// TwinCAT 3 PLC project PLCSim
// ProgramVersion: 3.1.4026.21
// libraries:
//   Tc2_Standard, * (Beckhoff Automation GmbH)
//   Tc2_System, * (Beckhoff Automation GmbH)
//   Tc3_Module, * (Beckhoff Automation GmbH)
//   VisuSymbols,newest,System
// project tree:
//   / GlobalTextList.TcGTLO, PlcTask.TcTTO (not stored), Visualization Manager.TcVMO (not stored)
//   POUs/ MAIN.TcPOU
//   VISUs/ Visualization.TcVIS
// real-time tasks:
//   TASK PlcTask: cycle T#30ms, priority 20, ADS port 350
// variable links:
//   PLCSim/PLCSim Instance <-> PLCStudent/PLCStudent Instance
//     PlcTask Inputs/MAIN.ixDrillDown <-> PlcTask Outputs/ControlFBD.qxDrillDown
//     PlcTask Inputs/MAIN.ixDrillUp <-> PlcTask Outputs/ControlFBD.qxDrillUp
//     PlcTask Inputs/MAIN.ixLampEmStopOk <-> PlcTask Outputs/ControlFBD.qxLampEmStopOk
//     PlcTask Inputs/MAIN.ixLampHomePos <-> PlcTask Outputs/ControlFBD.qxLampHomePos
//     PlcTask Inputs/MAIN.ixLampSafetyOk <-> PlcTask Outputs/ControlFBD.qxLampSafetyOk
//     PlcTask Inputs/MAIN.ixLampStarted <-> PlcTask Outputs/ControlFBD.qxLampStarted
//     PlcTask Inputs/MAIN.ixSliderAin <-> PlcTask Outputs/ControlFBD.qxSliderAin
//     PlcTask Inputs/MAIN.ixSliderAout <-> PlcTask Outputs/ControlFBD.qxSliderAout
//     PlcTask Inputs/MAIN.ixSliderBin <-> PlcTask Outputs/ControlFBD.qxSliderBin
//     PlcTask Inputs/MAIN.ixSliderBout <-> PlcTask Outputs/ControlFBD.qxSliderBout
//     PlcTask Outputs/MAIN.qxAuto <-> PlcTask Inputs/ControlFBD.ixAuto
//     PlcTask Outputs/MAIN.qxBtn1EmStopOk <-> PlcTask Inputs/ControlFBD.ixBtn1EmStopOk
//     PlcTask Outputs/MAIN.qxBtn2EmStopOk <-> PlcTask Inputs/ControlFBD.ixBtn2EmStopOk
//     PlcTask Outputs/MAIN.qxBtnAin <-> PlcTask Inputs/ControlFBD.ixBtnAin
//     PlcTask Outputs/MAIN.qxBtnAout <-> PlcTask Inputs/ControlFBD.ixBtnAout
//     PlcTask Outputs/MAIN.qxBtnBin <-> PlcTask Inputs/ControlFBD.ixBtnBin
//     PlcTask Outputs/MAIN.qxBtnBout <-> PlcTask Inputs/ControlFBD.ixBtnBout
//     PlcTask Outputs/MAIN.qxBtnDrillIn <-> PlcTask Inputs/ControlFBD.ixBtnDrillIn
//     PlcTask Outputs/MAIN.qxBtnDrillOut <-> PlcTask Inputs/ControlFBD.ixBtnDrillOut
//     PlcTask Outputs/MAIN.qxBtnReset <-> PlcTask Inputs/ControlFBD.ixBtnReset
//     PlcTask Outputs/MAIN.qxButtonStart <-> PlcTask Inputs/ControlFBD.ixButtonStart
//     PlcTask Outputs/MAIN.qxButtonStop <-> PlcTask Inputs/ControlFBD.ixButtonStop
//     PlcTask Outputs/MAIN.qxDrillDown <-> PlcTask Inputs/ControlFBD.ixDrillDown
//     PlcTask Outputs/MAIN.qxDrillUp <-> PlcTask Inputs/ControlFBD.ixDrillUp
//     PlcTask Outputs/MAIN.qxSafety1StopOk <-> PlcTask Inputs/ControlFBD.ixSafety1StopOk
//     PlcTask Outputs/MAIN.qxSafety2StopOk <-> PlcTask Inputs/ControlFBD.ixSafety2StopOk
//     PlcTask Outputs/MAIN.qxSliderAin <-> PlcTask Inputs/ControlFBD.ixSliderAin
//     PlcTask Outputs/MAIN.qxSliderAout <-> PlcTask Inputs/ControlFBD.ixSliderAout
//     PlcTask Outputs/MAIN.qxSliderBin <-> PlcTask Inputs/ControlFBD.ixSliderBin
//     PlcTask Outputs/MAIN.qxSliderBout <-> PlcTask Inputs/ControlFBD.ixSliderBout

// ---- POUs/MAIN.TcPOU
PROGRAM MAIN
VAR
	ixLampStarted	AT %I* : BOOL;
	ixSliderAout 	AT %I* : BOOL; 
	ixSliderAin 	AT %I* : BOOL; 
	ixSliderBout 	AT %I* : BOOL; 
	ixSliderBin 	AT %I* : BOOL; 
	ixDrillDown 	AT %I* : BOOL;
	ixDrillUp		AT %I* : BOOL;
	ixLampEmStopOk	AT %I* : BOOL;
	ixLampSafetyOk  AT %I* : BOOL;
	ixLampHomePos	AT %I* : BOOL;
	
	qxButtonStart	AT %Q* : BOOL;
	qxButtonStop	AT %Q* : BOOL;
	qxSliderAout	AT %Q* : BOOL;
	qxSliderAin		AT %Q* : BOOL;
	qxSliderBout	AT %Q* : BOOL;
	qxSliderBin		AT %Q* : BOOL;
	qxDrillUp		AT %Q* : BOOL;
	qxDrillDown		AT %Q* : BOOL;
	
	qxAuto			AT %Q* : BOOL;
	qxBtn1EmStopOk	AT %Q* : BOOL;
	qxBtn2EmStopOk	AT %Q* : BOOL;
	qxSafety1StopOk	AT %Q* : BOOL;
	qxSafety2StopOk	AT %Q* : BOOL;
	qxBtnReset  	AT %Q* : BOOL;
	qxBtnAout		AT %Q* : BOOL;
	qxBtnAin		AT %Q* : BOOL;
	qxBtnBout		AT %Q* : BOOL;
	qxBtnBin		AT %Q* : BOOL;
	qxBtnDrillOut	AT %Q* : BOOL;
	qxBtnDrillIn	AT %Q* : BOOL;
	mxReset 		: BOOL;
	mxCubeInvisible : BOOL;
	mxBtn1EmStop : BOOL;
	mxBtn2EmStop : BOOL;	
	
	nPosSliderA 	: INT:=0;
	nPosSliderB 	: INT:=0;
	nPosDrill 		: INT:=0;
	nPosXCube		: INT:=0;
	nPosYCube		: INT:=0;
	nSpeed 			: INT:=1;
	nCnt			: INT:=0;
	nErrorCnt		: INT:=0;
	nSeq: INT;
	
	fbTONAin:TON;
	fbTONAout:TON;
	fbTONBin:TON;
	fbTONBout:TON;
	fbTONDrillUp:TON;
	fbTONADrillDown:TON;
	
	
END_VAR

// Anders Nilsson 20230112

qxBtn1EmStopOk := NOT mxBtn1EmStop;
qxBtn2EmStopOk := NOT mxBtn2EmStop;

// Slider A
IF ixSliderAout AND NOT ixSliderAin THEN
	nPosSliderA := nPosSliderA-nSpeed;
	IF nPosSliderA < -75 THEN
		nPosSliderA := -75;
	END_IF
END_IF

IF ixSliderAin AND NOT ixSliderAout THEN
	nPosSliderA := nPosSliderA+nSpeed;
	IF nPosSliderA > 0 THEN
		nPosSliderA := 0;
	END_IF
END_IF

fbTONAin.PT := T#1S;
fbTONAin.IN := nPosSliderA = 0;
fbTONAin();
qxSliderAin := fbTONAin.Q;

fbTONAout.PT := T#1S;
fbTONAout.IN := nPosSliderA = -75;
fbTONAout();
qxSliderAout := fbTONAout.Q;



// Slider B
IF ixSliderBout AND NOT ixSliderBin THEN
	nPosSliderB := nPosSliderB + nSpeed;
	IF nPosSliderB > 0 THEN
		nPosSliderB := 0;
	END_IF
	
END_IF

IF ixSliderBin AND NOT ixSliderBout THEN
	nPosSliderB := nPosSliderB - nSpeed;
	IF nPosSliderB< -75 THEN
		nPosSliderB := -75;
	END_IF
END_IF

fbTONBin.PT := T#1S;
fbTONBin.IN := nPosSliderB = -75;
fbTONBin();
qxSliderBin := fbTONBin.Q;

fbTONBout.PT := T#1S;
fbTONBout.IN := nPosSliderB = 0;
fbTONBout();
qxSliderBout := fbTONBout.Q;




// Drill 
IF ixDrillDown AND NOT ixDrillUp THEN
	nPosDrill := nPosDrill + nSpeed;
	IF nPosDrill > 35 THEN
		nPosDrill := 35;
	END_IF
END_IF
	
IF ixDrillUp AND NOT ixDrillDown THEN
	nPosDrill := nPosDrill - nSpeed;
	IF nPosDrill < 0 THEN
		nPosDrill := 0;
	END_IF
END_IF
	
fbTONDrillUp.PT := T#1S;
fbTONDrillUp.IN := nPosDrill = 0;
fbTONDrillUp();
qxDrillUp := fbTONDrillUp.Q;

fbTONADrillDown.PT := T#1S;
fbTONADrillDown.IN := nPosDrill = 35;
fbTONADrillDown();
qxDrillDown := fbTONADrillDown.Q;


	
IF	mxReset THEN
	nSeq 		:= 10;
	nCnt 		:= 0;
	nErrorCnt   := 0;
	nPosSliderA := 0;
	nPosSliderB := 0;
	nPosDrill 	:= 0;
	nPosXCube   := 0;
	nPosYCube   := 0;
	mxCubeInvisible := FALSE;
END_IF
	

	
// Cube
CASE nSeq OF 
	0: 	//Start and Init Slider A in position
		IF 	qxSliderAIn THEN
			nPosXCube := 0;
		    nPosYCube := 0;
			mxCubeInvisible := FALSE;
			nSeq := 10;
		END_IF
		
	10:	//Slide A out
		nPosXCube := nPosSliderA;
		IF qxSliderAout THEN
			nSeq := 20;
		END_IF
		
		//Error
		IF  ixSliderAout AND ( NOT qxSliderBout OR NOT qxDrillUp) THEN
			nSeq := 100;
		END_IF
	
		
	20:	//Drill
	
		IF qxDrillDown THEN
			nSeq := 30;
		END_IF
		
		//Error
		IF 	NOT qxSliderAout OR NOT qxSliderBout  THEN
			nSeq := 100;
		END_IF
		
		
	30:  //Slide B in cube out
	
	    IF qxSliderBin AND NOT qxSliderAout THEN
			nCnt := nCnt +1;
			mxCubeInvisible := TRUE;
			nSeq := 0;
		END_IF
			
	100: //Error
		mxCubeInvisible := TRUE;
		IF 	qxSliderAIn THEN
			nErrorCnt := nErrorCnt +1;
			nSeq := 0;
		END_IF
	
	
END_CASE

END_PROGRAM

// ---- GlobalTextList.TcGTLO
TEXTLIST GlobalTextList
  791 = ' Exam Gr1'
  38 = ' Exam Gr1lant'
  498 = ' Exam Gr1Plant'
  372 = 'A'
  111 = 'Aut     Man'
  747 = 'Aut Man'
  923 = 'B'
  661 = 'Counter'
  201 = 'Counter %S'
  776 = 'Counter %s'
  882 = 'Counter %sCounter %s'
  833 = 'Cycle stop'
  36 = 'Cylibder B'
  529 = 'Cylibders B'
  223 = 'Cylinder A'
  735 = 'Cylinder B'
  726 = 'Drill'
  832 = 'Drill Plant'
  635 = 'Emergency stop'
  627 = 'Emergency Stop 1'
  511 = 'Emergency stop Ok'
  305 = 'Emergency Stop2'
  161 = 'Emergency Stop21'
  910 = 'Emergency stopOk'
  634 = 'Errors %s'
  556 = 'Home Pos'
  926 = 'In'
  848 = 'Manover'
  431 = 'Nilsson'
  255 = 'Nilsson\nzz'
  607 = 'Out'
  719 = 'Pusher'
  311 = 'Reset'
  659 = 'Reset safety'
  86 = 'Safety'
  758 = 'Safety \nGate'
  572 = 'Safety Gate'
  16 = 'Safety OK'
  761 = 'Slider A'
  571 = 'Slider B'
  532 = 'Start'
  609 = 'Start Auto'
  630 = 'Stop'
  348 = 'University West'
  517 = 'University West\nAnders Nilsson'
  245 = 'University West\nAnders Nilsson Nov 2019'
  193 = 'University West\nAnders Nilsson Nov 2022'
  486 = 'University West\nAnders Nilsson Nov 2023'
END_TEXTLIST

// ---- VISUs/Visualization.TcVIS
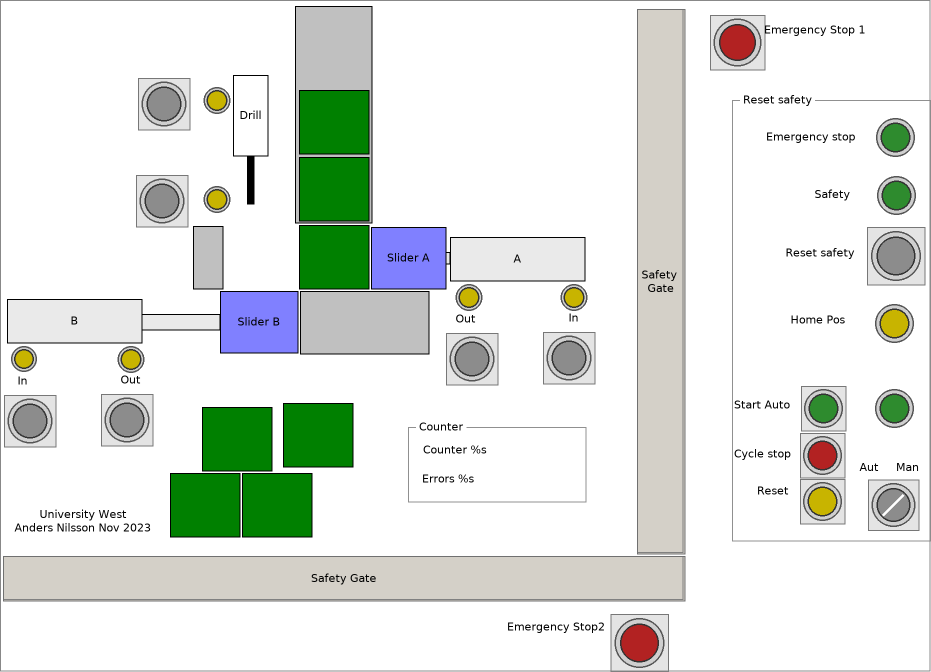
VISUALIZATION Visualization  // 931x672
    Group (233,75 59x138)
        p2773130477: main.nPosDrill
        p1126004900: MAIN.nPosDrill
        Rectangle (0,0 35x81), "Drill"
        Rectangle (14,81 7x48)
    Rectangle (295,6 77x217)
    Rectangle (299,225 70x64), invisible if: MAIN.mxCubeInvisible
        p3528305787: MAIN.nPosXCube
        p874137650: MAIN.nPosXCube
        p2773130477: MAIN.nPosYCube
        p1126004900: MAIN.nPosYCube
    Rectangle (193,226 30x63)
    Rectangle (299,157 70x64)
    Rectangle (300,291 129x63)
    Rectangle (299,90 70x64)
    Lamp1 (115,344 32x31), variable: MAIN.qxSliderBout, style: Lamp-Lamp1-Yellow
    Lamp1 (8,344 32x30), variable: MAIN.qxSliderBin, style: Lamp-Lamp1-Yellow
    Lamp1 (558,282 32x31), variable: MAIN.qxSliderAin, style: Lamp-Lamp1-Yellow
    Lamp1 (453,282 32x31), variable: MAIN.qxSliderAout, style: Lamp-Lamp1-Yellow
    Lamp1 (201,85 32x31), variable: MAIN.qxDrillUp, style: Lamp-Lamp1-Yellow
    Lamp1 (201,184 32x31), variable: MAIN.qxDrillDown, style: Lamp-Lamp1-Yellow
    Rectangle (242,473 70x64), invisible if: main.nCnt < 1
    Rectangle (283,403 70x64), invisible if: main.nCnt < 4
    Rectangle (170,473 70x64), invisible if: main.nCnt < 2
    Rectangle (202,407 70x64), invisible if: main.nCnt < 3
    GroupBox (732,92 199x449), "Reset safety"
        Label (0,290 60x46), "Start Auto"
        PushSwitch (69,294 45x45), variable: MAIN.qxButtonStart, behaviour: TAP, style: Switch-PushSwitch-Green
        PushSwitch (68,341 45x45), variable: MAIN.qxButtonStop, behaviour: TAP, style: Switch-PushSwitch-Red
        Lamp1 (140,294 45x45), variable: MAIN.ixLampStarted, style: Lamp-Lamp1-Green
        Label (0,339 61x46), "Cycle stop"
        Label (50,133 76x56), "Reset safety"
        PushSwitch (135,134 58x60), variable: MAIN.qxBtnReset, behaviour: TAP, style: Switch-PushSwitch-Gray
        Label (75,88 51x29), "Safety"
        Label (32,17 94x56), "Emergency stop"
        Lamp1 (141,23 45x45), variable: MAIN.ixLampEmStopOk, style: Lamp-Lamp1-Green
        Lamp1 (142,81 45x45), variable: MAIN.ixLampSafetyOk, style: Lamp-Lamp1-Green
        RotarySwitch (136,386 51x54), variable: MAIN.qxAuto, behaviour: TOGGLE, style: Switch-RotarySwitch-Gray
        Label (121,362 73x27), "Aut Man"
        Lamp1 (140,209 45x45), variable: MAIN.ixLampHomePos, style: Lamp-Lamp1-Yellow
        Label (48,200 76x56), "Home Pos"
        Label (20,376 42x46), "Reset"
        PushSwitch (68,387 45x45), variable: MAIN.mxReset, behaviour: TAP, style: Switch-PushSwitch-Yellow
    GroupBox (408,419 178x83), "Counter"
        Rectangle (12,16 112x30), "Counter %s", text variable: MAIN.nCnt
        Rectangle (11,45 112x30), "Errors %s", text variable: MAIN.nErrorCnt
    Label (447,302 37x34), "Out"
    Label (112,363 37x34), "Out"
    Label (555,301 37x34), "In"
    Label (4,364 37x34), "In"
    Rectangle (371,252 79x12)
    Rectangle (450,237 135x44), "A"
    Rectangle (139,314 81x16)
    Rectangle (7,299 135x44), "B"
    Rectangle (371,227 75x62), "Slider A"
        p3528305787: MAIN.nPosSliderA
        p874137650: MAIN.nPosSliderA
    Rectangle (220,291 78x62), "Slider B"
        p3528305787: MAIN.nPosSliderB
        p874137650: MAIN.nPosSliderB
    Label (7,500 152x42), "University West Anders Nilsson Nov 2023"
    PushSwitch (446,332 52x54), variable: MAIN.qxBtnAout, behaviour: TAP, style: Switch-PushSwitch-Gray
    PushSwitch (543,331 52x54), variable: MAIN.qxBtnAin, behaviour: TAP, style: Switch-PushSwitch-Gray
    PushSwitch (101,393 52x54), variable: MAIN.qxBtnBout, behaviour: TAP, style: Switch-PushSwitch-Gray
    PushSwitch (4,394 52x54), variable: MAIN.qxBtnBin, behaviour: TAP, style: Switch-PushSwitch-Gray
    PushSwitch (136,174 52x54), variable: MAIN.qxBtnDrillOut, behaviour: TAP, style: Switch-PushSwitch-Gray
    PushSwitch (138,77 52x54), variable: MAIN.qxBtnDrillIn, behaviour: TAP, style: Switch-PushSwitch-Gray
    PushSwitch (703,15 69x55), variable: MAIN.mxBtn1EmStop, behaviour: TOGGLE, style: Switch-PushSwitch-Red
    Button (637,9 48x545), "Safety Gate"
        toggle MAIN.qxSafety1StopOk
    PushSwitch (606,614 67x58), variable: MAIN.mxBtn2EmStop, behaviour: TOGGLE, style: Switch-PushSwitch-Red
    Button (3,556 682x45), "Safety Gate"
        toggle MAIN.qxSafety2StopOk
    Label (745,2 140x56), "Emergency Stop 1"
    Label (486,599 140x56), "Emergency Stop2"
END_VISUALIZATION
